{attribute 'linkalways'} 
{attribute 'no_explicit_call' := 'This FB is a CLASS and must be accessed using methods or properties'}
{attribute 'enable_dynamic_creation'}
FUNCTION_BLOCK CreateGraphRpcHandler IMPLEMENTS I_AsynchronousRpcHandler
VAR
	graphFramework : I_GraphFramework;
	graphs : I_Graphs;
	lastGraphUuid : T_MAXSTRING;
END_VAR

METHOD Handle
VAR_INPUT
	Parameters : I_Deserializer;
	Response : I_AsynchronousRpcResponse;
END_VAR
VAR
	graph : I_Graph;
	feedback : DeserializerFeedback;
	graphDeserializer : I_Deserializer;
	serializer : I_Serializer;
	getStatusVisitor : GetStatusVisitor;
END_VAR
IF graphs.TryGetGraphByUuid(lastGraphUuid, graph) THEN
	graphs.RemoveGraph(graph);
	graph.Dispose();
	lastGraphUuid := '';
END_IF

graph := graphFramework.Create();
graphDeserializer := Parameters.GetKeyObject('graph');

IF NOT graph.TryDeserializeFrom(graphDeserializer, feedback) THEN
	Response.RejectWithMessage(feedback.FirstError.Message);
	graph.Dispose();
	RETURN;
END_IF

lastGraphUuid := graph.Uuid;
graphs.AddGraph(graph);

serializer := Response.GetSerializer();
getStatusVisitor.Initialize(serializer);
getStatusVisitor.VisitGraph(graph);
Response.CompleteWithSerializer(serializer);
serializer.Dispose();
END_METHOD

METHOD PUBLIC Initialize
VAR_INPUT
	GraphFramework : I_GraphFramework;
	Graphs : I_Graphs;
END_VAR
THIS^.graphFramework := GraphFramework;
THIS^.graphs := Graphs;
END_METHOD

END_FUNCTION_BLOCK

(* stored: Version 1.1.0.1, ProductVersion 3.1.4024.13
   POU CreateGraphRpcHandler: Id {40b56d4c-0583-457f-b6b7-cb5e579f4531}, SpecialFunc None
   Method Handle: Id {7b2ef4f3-c265-4943-8044-4e6d6c3e0273}
   Method Initialize: Id {6f5caa5d-c012-44e1-8933-f5f8ca304953} *)
